Universal Robots PolyScope program: Ejercicio_2.urp

Program Ejercicio_2 (installation=default directory=/home/ur/ursim-current/programs/Ejercicio_2 createdIn=5.7.0.90932 lastSavedIn=5.7.0.90932 robotSerialNumber=20195599999)
Calibrated DH parameters: a=[0, -0.425, -0.3922, 0, 0, 0]; d=[0.1625, 0, 0, 0.1333, 0.0997, 0.0996]; alpha=[1.570796, 0, 0, 1.570796, -1.570796, 0]; deltaTheta=[0, 0, 0, 0, 0, 0]
Robot Program (runOnlyOnce=true)
  Script file /home/ur/ursim-current/programs/Ejercicio_2/Ejercicio_2.script
    | # Preparar instalacion
    | set_gravity([0,0,9.8])
    | set_tcp(p[0,0.025,0.175,0,0,1.57])
    | set_payload_mass(2)
    | 
    | # Variables
    | varx = 0
    | vary = 0
    | n_filas = 2.0
    | n_columnas = 2.0
    | d_filas = 0.02
    | d_columnas = 0.02
    | i=0
    | j=0
    | 
    | #rutina de desbarbado
    | def desbarbado(varx, vary, n_filas, n_columnas, d_filas, d_columnas):
    |  set_digital_out(0,True)
    |  while i < n_columnas:
    |   while  j < n_filas:
    |    pose_pre = p[0.5+varx,-0.150+vary,0.05,0,3.1416,0]
    |    pose_desb = p[0.5+varx,-0.150+vary,0,0,3.1416,0]
    |    movej(pose_pre,1.5,1) #acercamiento
    |    movel(pose_desb,1.5,1) #punto desbarbado
    |    sleep(2.5)
    |    movej(pose_pre,1.5,1) #salida
    |    varx=varx+d_filas
    |    i=i+1
    |   end
    |  varx=0
    |  i=0
    |  vary=vary+d_columnas
    |  j=j+1
    | end
    | set_digital_out(0,False)
    | end
    | 
    | #Programa
    | popup("Iniciando programa desbarbado rejillas",title="Titulo",warning=False,blocking=True)
    | textmsg("Iniciando programa")
    | safe_pose = [0,-0.78,-1.57,-2.35,1.57,0]
    | movej(safe_pose,1.5,1)
    | desbarbado (varx, vary, n_filas, n_columnas, d_filas, d_columnas)
    | movej(safe_pose,1.5,1)
